PROGRAM PRG_TEST
VAR
	// Test suite instances
	fbCommandTest : FB_ST_HMICommand_Test;
	fbComponentAPITest : FB_ST_HMIComponentAPI_Test;
	fbStatusTest : FB_ST_HMIStatus_Test;
	fbHMIBaseTest : FB_HMIBase_Test;
END_VAR

// ============================================================================
// UiBuilder Library Test Suite
// ============================================================================
// This program runs all unit tests for the UiBuilder library using TcUnit
// framework. Call this program from your main task to execute tests.
//
// Test Coverage:
// - ST_HMICommand data type tests
// - ST_HMIComponentAPI data type tests
// - ST_HMIStatus data type tests
// - FB_HMIBase function block tests
//
// Usage:
// 1. Add PRG_TEST to your PlcTask or call from MAIN
// 2. Build and download the project
// 3. Run the PLC
// 4. Check TcUnit results in the output window
// ============================================================================

// Execute all test suites
// TcUnit automatically collects and reports results through FB_TestSuite base class
fbCommandTest();
fbComponentAPITest();
fbStatusTest();
fbHMIBaseTest();

END_PROGRAM

(* stored: Version 1.1.0.1
   POU PRG_TEST: Id {a5555555-5555-5555-5555-555555555555}, SpecialFunc None *)
